PROGRAM Step
VAR
	PreviousStepComplete: BOOL;
	StepDone: BOOL;
	StepComplete: BOOL;
	StepInProgress: BOOL;
	SequenceStart: BOOL;
	CylinderExtended: BOOL;
	Step1Complete: BOOL;
	Step1InProgress: BOOL;
	CylinderRetracted: BOOL;
	Step2Complete: BOOL;
	Step2InProgress: BOOL;
	SequenceComplete: BOOL;
END_VAR

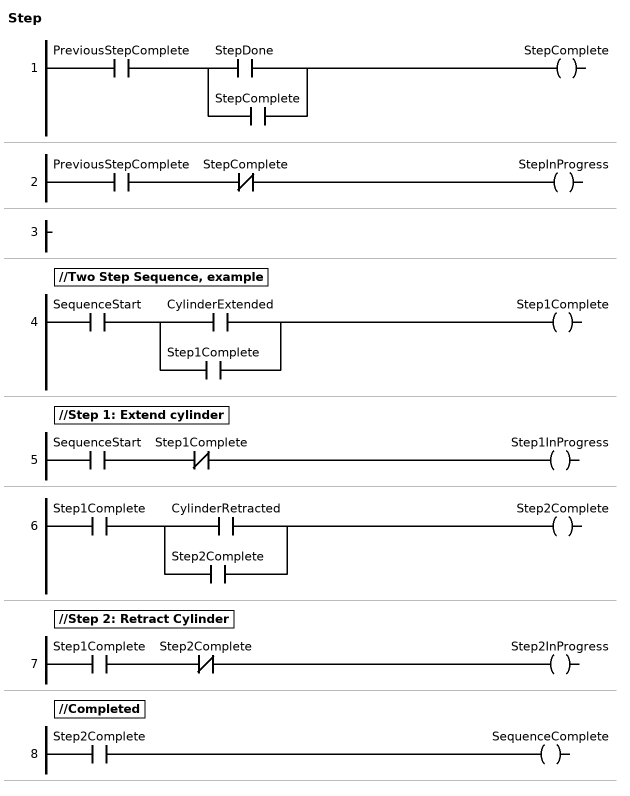
// NETWORK 1
StepComplete := PreviousStepComplete AND (StepDone OR StepComplete);

// NETWORK 2
StepInProgress := PreviousStepComplete AND NOT StepComplete;

// NETWORK 3

// NETWORK 4
// label: //Two Step Sequence, example
Step1Complete := SequenceStart AND (CylinderExtended OR Step1Complete);

// NETWORK 5
// label: //Step 1: Extend cylinder
Step1InProgress := SequenceStart AND NOT Step1Complete;

// NETWORK 6
Step2Complete := Step1Complete AND (CylinderRetracted OR Step2Complete);

// NETWORK 7
// label: //Step 2: Retract Cylinder
Step2InProgress := Step1Complete AND NOT Step2Complete;

// NETWORK 8
// label: //Completed
SequenceComplete := Step2Complete;

END_PROGRAM

(* stored: Version 1.1.0.1, ProductVersion 3.1.4024.10
   POU Step: Id {82d3a960-5bfd-4606-a664-5fe9bc8eb5cc}, SpecialFunc None *)
